PROGRAM PRG_GetSystemTime
VAR_OUTPUT
	sQTime:	TIMESTRUCT;	(* Output: Timeinformation *)
END_VAR
VAR
	fbNTGetTime:	NT_GetTime;
	fbTONGetTime:	TON;
END_VAR


(* Receive the NT-Time every second *)
fbTONGetTime( IN := TRUE, PT := T#1s );
IF fbTONGetTime.Q THEN
	fbNTGetTime( START := FALSE );
	fbTONGetTime( IN := FALSE );
END_IF
fbNTGetTime
	(	START := TRUE,
		TMOUT := DEFAULT_ADS_TIMEOUT
	);

(* Setting the result *)
sQTime	:= fbNTGetTime.TIMESTR;

END_PROGRAM

(* stored: Version 1.1.0.1, ProductVersion 3.1.4024.9
   POU PRG_GetSystemTime: Id {560fbe79-d00e-4e7a-9889-60fb936bcbb6}, SpecialFunc None *)
